# EPICS substitutions: iocs/miroTest/miroTestApp/Db/miroCamera.substitutions
file miroCamera.template {
pattern{ P, R , PORT, ADDR, TIMEOUT}
{ "test:", "ioc:" , "MIRO", 0, 1}
}
